FUNCTION_BLOCK SERVER_2_3 (* Generic server (2 SD, 3 RD); instantiated from GEN_SERVER *)
  (* Standard: 61499-2 *)
  (* Version 0.1, 2026-09-28, Project contributors, AAU Smart Production Lab *)
  PACKAGE iec61499::net;
  {SET_ATTRIBUTE(eclipse4diac::core::GenericClassName, 'GEN_SERVER')}
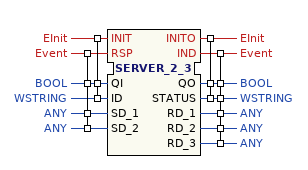
  EVENT_INPUT
    INIT : EInit WITH QI, ID;
    RSP WITH QI, SD_1, SD_2;
  END_EVENT
  EVENT_OUTPUT
    INITO : EInit WITH QO, STATUS;
    IND WITH QO, STATUS, RD_1, RD_2, RD_3;
  END_EVENT
  VAR_INPUT
    QI : BOOL;
    ID : WSTRING;
    SD_1 : ANY;
    SD_2 : ANY;
  END_VAR
  VAR_OUTPUT
    QO : BOOL;
    STATUS : WSTRING;
    RD_1 : ANY;
    RD_2 : ANY;
    RD_3 : ANY;
  END_VAR
END_FUNCTION_BLOCK
